FUNCTION_BLOCK TwoConCtlMulticast (* Composite Function Block Type *)
  (* Standard: 61499-2 *)
  (* Version 0.2, 2003-12-05, JHC, Rockwell Automation, Renamed from NEWCOMPFB. *)
  (* Version 0.1, 2002-01-08, JHC, Rockwell Automation, Added DLY FB as example. *)
  (* Version 0.0, 2000-05-27, JHC, Rockwell Automation *)
  (* Compiler header: package fb.rt.cs725; *)
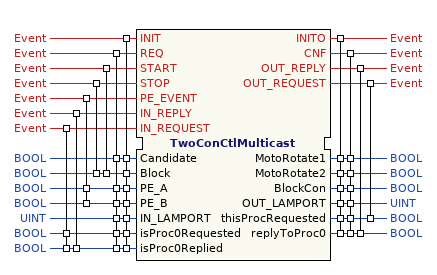
  EVENT_INPUT
    INIT WITH Candidate, Block, PE_A, PE_B, IN_LAMPORT, isProc0Requested, isProc0Replied; (* Initialization Request *)
    REQ WITH Candidate, PE_A, PE_B, IN_LAMPORT, isProc0Requested, isProc0Replied; (* Normal Execution Request *)
    START WITH Block;
    STOP WITH Block;
    PE_EVENT WITH PE_A, PE_B;
    IN_REPLY WITH isProc0Replied;
    IN_REQUEST WITH isProc0Requested, isProc0Replied;
  END_EVENT
  EVENT_OUTPUT
    INITO WITH MotoRotate1, MotoRotate2, BlockCon, OUT_LAMPORT, thisProcRequested, replyToProc0; (* Initialization Confirm *)
    CNF WITH MotoRotate1, MotoRotate2, BlockCon, OUT_LAMPORT, thisProcRequested, replyToProc0; (* Execution Confirmation *)
    OUT_REPLY WITH replyToProc0;
    OUT_REQUEST WITH thisProcRequested;
  END_EVENT
  VAR_INPUT
    Candidate : BOOL;
    Block : BOOL;
    PE_A : BOOL;
    PE_B : BOOL;
    IN_LAMPORT : UINT;
    isProc0Requested : BOOL;
    isProc0Replied : BOOL;
  END_VAR
  VAR_OUTPUT
    MotoRotate1 : BOOL;
    MotoRotate2 : BOOL;
    BlockCon : BOOL;
    OUT_LAMPORT : UINT;
    thisProcRequested : BOOL;
    replyToProc0 : BOOL;
  END_VAR
  FBS
    FC11 : ConveyorCTL(Candidate := 0, Block := 0);
    FC12 : ConveyorCTLMulticast;
  END_FBS
  EVENT_CONNECTIONS
    INIT TO FC11.INIT;
    REQ TO FC11.REQ;
    FC12.INITO TO INITO;
    FC12.CNF TO CNF;
    REQ TO FC12.REQ;
    STOP TO FC12.CAS_STOP;
    START TO FC12.CAS_START;
    FC12.STOP TO FC11.CAS_STOP;
    FC12.START TO FC11.CAS_START;
    FC11.INITO TO FC12.INIT;
    PE_EVENT TO FC12.PE_EVENT;
    IN_REPLY TO FC12.IN_REPLY;
    IN_REQUEST TO FC12.IN_REQUEST;
    FC12.OUT_REPLY TO OUT_REPLY;
    FC12.OUT_REQUEST TO OUT_REQUEST;
  END_CONNECTIONS
  DATA_CONNECTIONS
    Block TO FC12.Block;
    Candidate TO FC12.Candidate;
    FC12.BlockCon TO BlockCon;
    FC11.MotoRotate TO MotoRotate1;
    FC12.MotoRotate TO MotoRotate2;
    PE_B TO FC11.PE;
    PE_A TO FC12.PE_IN;
    PE_B TO FC12.PE_OUT;
    IN_LAMPORT TO FC12.IN_LAMPORT;
    FC12.OUT_LAMPORT TO OUT_LAMPORT;
    FC12.thisProcRequested TO thisProcRequested;
    FC12.replyToProc0 TO replyToProc0;
    isProc0Requested TO FC12.isProc0Requested;
    isProc0Replied TO FC12.isProc0Replied;
  END_CONNECTIONS
END_FUNCTION_BLOCK
